// TIA Portal V19 export
TYPE "LEXCHANGETRAY_typeConstraintRollerEm_toConstraintWorkstationReq"
// stored: Access Published
   STRUCT
      transferEnable : Bool;   // 请求转移
      unConstraint : Bool;
      Constraint : Bool;
   END_STRUCT;
END_TYPE
